TYPE ST_HTTP_Response :
STRUCT
	arrHeaders	: ARRAY [0..HTTP_RESPONSE_HEADER_ARRAY_SIZE] OF STRING;
	sContent	: STRING(255);
END_STRUCT
END_TYPE

(* stored: Version 1.1.0.1, ProductVersion 3.1.4020.12
   DUT ST_HTTP_Response: Id {364ca746-f841-4792-9336-b774ccbe37fe} *)
